(* PLC project CoDeSys External Library Template, WAGO e!COCKPIT e!COCKPIT, author 3S - Smart Software Solutions GmbH *)
(* stored: creationDateTime 2019-10-29T12:22:40.6747974, version 3.5.5.30, modificationDateTime 2019-10-24T14:40:07.960949, organization 3S - Smart Software Solutions GmbH *)
(* Library project template with all possible element types, docu and a sample project structure *)

FUNCTION_BLOCK fbPPPSBramkaSTC65RS485Modbus
  VAR_INPUT
    sKomunikat : alSTRINGKomunikat;  (* komunikat z systemu zewnętrznego *)
    intTablicaKomunikatowRozmiar : INT;  (* rozmiar tablicy danych wysyłkowych *)
    xTablicaKomunikatowHold : BOOL;  (* wstrzymanie komunikacji mniej ważnych komunikatów *)
    sIdInstancji : STRING;  (* parametr ID rolety np NS02L*202IBM**** *)
    sIdAplikacji : STRING;  (* parametr ID aplikacji np SO*******ECL*000 *)
    sMnemonik : STRING;  (* mnemonik właściciela - BCB* *)
    sMACAdres : STRING;  (* MAC adres sterownika *)
    sDaneZapasowe : STRING;  (* 6 znaków zapasu *)
    tCzasOpoznieniaRestartu : TIME;  (* czas opóźnienia po którym zaczynają być raportowane wartości *)
    bAdres : BYTE;
    tMinimalnyCzasRaportowania : TIME;
    tMaksymalnyCzasRaportowania : TIME;
    tCzasTimeoutEnOcean : TIME;
  END_VAR
  VAR_IN_OUT
    arModbusStatusKomunikacji : ARRAY[1..256] OF INT;
    arModbusOdczytCykliczny : ARRAY[1..5000] OF typModbusOdczytCykliczny;
    arTablicaKomunikatow : alARRAYTablicaKomunikatow;
    intTablicaKomunikatowZnacznikZapisu : INT;
  END_VAR
  VAR CONSTANT
    wCzasDzialaniaOdResetuAlarm : WORD := 120;
  END_VAR
  VAR
    xPierwszySkan : BOOL := TRUE;
    intPetlaPierwszySkan : INT := 1;
    xPoInicjalizacji : BOOL := FALSE;  (* inicjalizacja *)
    fbInicjalizacyjnyTimer : TON;
    uintFirmwareVersion : UINT := 0;  (* definicja adresów i zmiennych modbusowych *)
    wFirmwareVersion : WORD;
    uintOperatingTimeSinceLastResetHi : UINT := 2;
    wOperatingTimeSinceLastResetHi : WORD;
    uintOperatingTimeSinceLastResetLo : UINT := 3;
    wOperatingTimeSinceLastResetLo : WORD;
    uintReceivingChannelsTelegramCounterAllIDsHi : UINT := 4;
    wReceivingChannelsTelegramCounterAllIDsHi : WORD;
    uintReceivingChannelsTelegramCounterAllIDsLo : UINT := 5;
    wReceivingChannelsTelegramCounterAllIDsLo : WORD;
    uintReceivingChannelsTelegramCounterStoredIDsHi : UINT := 6;
    wReceivingChannelsTelegramCounterStoredIDsHi : WORD;
    uintReceivingChannelsTelegramCounterStoredIDsLo : UINT := 7;
    wReceivingChannelsTelegramCounterStoredIDsLo : WORD;
    uintEnOceanBaseIdByte3 : UINT := 8;
    wEnOceanBaseIdByte3 : WORD;
    uintEnOceanBaseIdByte2 : UINT := 9;
    wEnOceanBaseIdByte2 : WORD;
    uintEnOceanBaseIdByte1 : UINT := 10;
    wEnOceanBaseIdByte1 : WORD;
    uintEnOceanBaseIdByte0 : UINT := 11;
    wEnOceanBaseIdByte0 : WORD;
    uintRepeaterFunction : UINT := 15;
    wRepeaterFunction : WORD;
    uintMinResponseTime : UINT := 16;
    wMinResponseTime : WORD;
    uintResetRxCoil : UINT := 17;
    wResetRxCoil : WORD;
    uintTransmittingChannelsTelegramCounterAll : UINT := 18;
    wTransmittingChannelsTelegramCounterAll : WORD;
    uintTransmittingChannelsTelegramCounterByCoilTriggered : UINT := 19;
    wTransmittingChannelsTelegramCounterByCoilTriggered : WORD;
    wCzasDzialaniaOdResetuHi : WORD;  (* zmienne operacyjne Zmienne Modbusowe *)
    wCzasDzialaniaOdResetuLo : WORD;
    dwCzasDzialaniaOdResetu : DWORD;
    xAlarmResetu : BOOL;
    wLicznikTelegramowUrzadzenHi : WORD;
    wLicznikTelegramowUrzadzenLo : WORD;
    dwLicznikTelegramowUrzadzen : DWORD;
    dwLicznikTelegramowUrzadzenPamiec : DWORD;
    fbTimeoutEnOcean : TON;
    wFunkcjaPowtarzanaia : WORD;
    wMinimalnyCzasOdpowiedzi : WORD;
    sDane : alSTRINGKomunikat;
    sWyslanyKomunikat : alSTRINGKomunikat;
    sKomunikatPamiec : alSTRINGKomunikat;
    sWyslanyKomunikatDummy : alSTRINGKomunikat;
    intPetla : INT;
    arErrorStan : ARRAY[0..5] OF INT;  (* tablica przechowująca statusy alarmowe *)
    arErrorKlasa : ARRAY[0..5] OF INT;  (* tablica przechowująca klasy danych alarmów *)
    fbBrakKomunikacjiTimer : TON;  (* Wystawianie alarmu o braku komunikacji. Alarm zostanie aktywowany po minutach od momentu stwierdzenia braku komunikacji. *)
  END_VAR

            (*			
Autor:					Paweł Kąkol, 2018-08-13, Jan Bartczak
Prawa majątkowe: 		Solwena Sp. z o.o., 
Aktualizacje:			
						
Opis:					fb służy obsługi bramek (STC65-RS485) GTW0 na budynkach PPP Sopot (ENGIE) 
		
UWAGA:					2018-08-13-PK-Stworzenie FB
						2018-10-05-JB Przygotowanie odczytu rejestrów Modbusowych z bramki STC
						2018-12-11-JB Poprawienie obsługi alarmów od resetu bramki i braku ruchu telegramów (do tego momentu wysyłane były błędne alarmy)		
						2019-02-18-AWy: Filtrowanie alarmu braku komunikacji (5 minut zwłoki od momentu stwierdzenia braku komunikacji)			
*)

//inicjalizacja sterownika
fbInicjalizacyjnyTimer(IN := NOT xPoInicjalizacji , PT := tCzasOpoznieniaRestartu);
IF fbInicjalizacyjnyTimer.Q THEN
	xPoInicjalizacji := TRUE;
	dwLicznikTelegramowUrzadzenPamiec := dwLicznikTelegramowUrzadzen;
END_IF


IF xPierwszySkan THEN
	xPierwszySkan := FALSE;
	WHILE arModbusOdczytCykliczny[intPetlaPierwszySkan].bAdresUrzadzenia <> 0 DO
		intPetlaPierwszySkan := intPetlaPierwszySkan + 1;
	END_WHILE
	
//deklaracja rejestrow do odczytu

	//wyznaczenie adresów rejestrów modbusowych

	//holding register
	//  #Firmware Version e.g.: 0x3300 = Version 3.3.0.0
	arModbusOdczytCykliczny[intPetlaPierwszySkan].bAdresUrzadzenia := bAdres;
	arModbusOdczytCykliczny[intPetlaPierwszySkan].bFunkcja := TO_BYTE(enumModbusKodyFunkcji.OdczytNRejestrow);
	arModbusOdczytCykliczny[intPetlaPierwszySkan].uiAdresRejestru := uintFirmwareVersion;
	arModbusOdczytCykliczny[intPetlaPierwszySkan].ltCzestotliwosc := TIME_TO_LTIME(tMinimalnyCzasRaportowania);
	arModbusOdczytCykliczny[intPetlaPierwszySkan].pZmiennaReferencyjna := ADR(wFirmwareVersion);
	intPetlaPierwszySkan := intPetlaPierwszySkan + 1;

	//R/W Operating Time since last reset [seconds] HIGH
	arModbusOdczytCykliczny[intPetlaPierwszySkan].bAdresUrzadzenia := bAdres;
	arModbusOdczytCykliczny[intPetlaPierwszySkan].bFunkcja := TO_BYTE(enumModbusKodyFunkcji.OdczytNRejestrow);
	arModbusOdczytCykliczny[intPetlaPierwszySkan].uiAdresRejestru := uintOperatingTimeSinceLastResetHi;
	arModbusOdczytCykliczny[intPetlaPierwszySkan].ltCzestotliwosc := TIME_TO_LTIME(tMinimalnyCzasRaportowania);
	arModbusOdczytCykliczny[intPetlaPierwszySkan].pZmiennaReferencyjna := ADR(wOperatingTimeSinceLastResetHi);
	intPetlaPierwszySkan := intPetlaPierwszySkan + 1;	
	
	//R/W Operating Time since last reset [seconds] LOW
	arModbusOdczytCykliczny[intPetlaPierwszySkan].bAdresUrzadzenia := bAdres;
	arModbusOdczytCykliczny[intPetlaPierwszySkan].bFunkcja := TO_BYTE(enumModbusKodyFunkcji.OdczytNRejestrow);
	arModbusOdczytCykliczny[intPetlaPierwszySkan].uiAdresRejestru := uintOperatingTimeSinceLastResetLo;
	arModbusOdczytCykliczny[intPetlaPierwszySkan].ltCzestotliwosc := TIME_TO_LTIME(tMinimalnyCzasRaportowania);
	arModbusOdczytCykliczny[intPetlaPierwszySkan].pZmiennaReferencyjna := ADR(wOperatingTimeSinceLastResetLo);
	intPetlaPierwszySkan := intPetlaPierwszySkan + 1;	
	
	//R/W Receiving Channels Telegram Counter (all IDs) HIGH
	arModbusOdczytCykliczny[intPetlaPierwszySkan].bAdresUrzadzenia := bAdres;
	arModbusOdczytCykliczny[intPetlaPierwszySkan].bFunkcja := TO_BYTE(enumModbusKodyFunkcji.OdczytNRejestrow);
	arModbusOdczytCykliczny[intPetlaPierwszySkan].uiAdresRejestru := uintReceivingChannelsTelegramCounterAllIDsHi;
	arModbusOdczytCykliczny[intPetlaPierwszySkan].ltCzestotliwosc := TIME_TO_LTIME(tMinimalnyCzasRaportowania);
	arModbusOdczytCykliczny[intPetlaPierwszySkan].pZmiennaReferencyjna := ADR(wReceivingChannelsTelegramCounterAllIDsHi);
	intPetlaPierwszySkan := intPetlaPierwszySkan + 1;		

	//R/W Receiving Channels Telegram Counter (all IDs) LOW	
	arModbusOdczytCykliczny[intPetlaPierwszySkan].bAdresUrzadzenia := bAdres;
	arModbusOdczytCykliczny[intPetlaPierwszySkan].bFunkcja := TO_BYTE(enumModbusKodyFunkcji.OdczytNRejestrow);
	arModbusOdczytCykliczny[intPetlaPierwszySkan].uiAdresRejestru := uintReceivingChannelsTelegramCounterAllIDsLo;
	arModbusOdczytCykliczny[intPetlaPierwszySkan].ltCzestotliwosc := TIME_TO_LTIME(tMinimalnyCzasRaportowania);
	arModbusOdczytCykliczny[intPetlaPierwszySkan].pZmiennaReferencyjna := ADR(wReceivingChannelsTelegramCounterAllIDsLo);
	intPetlaPierwszySkan := intPetlaPierwszySkan + 1;

	//R/W Receiving Channels Telegram Counter (stored IDs only) HIGH
	arModbusOdczytCykliczny[intPetlaPierwszySkan].bAdresUrzadzenia := bAdres;
	arModbusOdczytCykliczny[intPetlaPierwszySkan].bFunkcja := TO_BYTE(enumModbusKodyFunkcji.OdczytNRejestrow);
	arModbusOdczytCykliczny[intPetlaPierwszySkan].uiAdresRejestru := uintReceivingChannelsTelegramCounterStoredIDsHi;
	arModbusOdczytCykliczny[intPetlaPierwszySkan].ltCzestotliwosc := TIME_TO_LTIME(tMinimalnyCzasRaportowania);
	arModbusOdczytCykliczny[intPetlaPierwszySkan].pZmiennaReferencyjna := ADR(wReceivingChannelsTelegramCounterStoredIDsHi);
	intPetlaPierwszySkan := intPetlaPierwszySkan + 1;

	//R/W Receiving Channels Telegram Counter (stored IDs only) LOW
	arModbusOdczytCykliczny[intPetlaPierwszySkan].bAdresUrzadzenia := bAdres;
	arModbusOdczytCykliczny[intPetlaPierwszySkan].bFunkcja := TO_BYTE(enumModbusKodyFunkcji.OdczytNRejestrow);
	arModbusOdczytCykliczny[intPetlaPierwszySkan].uiAdresRejestru := uintReceivingChannelsTelegramCounterStoredIDsLo;
	arModbusOdczytCykliczny[intPetlaPierwszySkan].ltCzestotliwosc := TIME_TO_LTIME(tMinimalnyCzasRaportowania);
	arModbusOdczytCykliczny[intPetlaPierwszySkan].pZmiennaReferencyjna := ADR(wReceivingChannelsTelegramCounterStoredIDsLo);
	intPetlaPierwszySkan := intPetlaPierwszySkan + 1;	
	
	//R/W* #EnOcean Base-ID-Byte-3
	arModbusOdczytCykliczny[intPetlaPierwszySkan].bAdresUrzadzenia := bAdres;
	arModbusOdczytCykliczny[intPetlaPierwszySkan].bFunkcja := TO_BYTE(enumModbusKodyFunkcji.OdczytNRejestrow);
	arModbusOdczytCykliczny[intPetlaPierwszySkan].uiAdresRejestru := uintEnOceanBaseIdByte3;
	arModbusOdczytCykliczny[intPetlaPierwszySkan].ltCzestotliwosc := TIME_TO_LTIME(tMinimalnyCzasRaportowania);
	arModbusOdczytCykliczny[intPetlaPierwszySkan].pZmiennaReferencyjna := ADR(wEnOceanBaseIdByte3);
	intPetlaPierwszySkan := intPetlaPierwszySkan + 1;	
	
	//R/W* #EnOcean Base-ID-Byte-2
	arModbusOdczytCykliczny[intPetlaPierwszySkan].bAdresUrzadzenia := bAdres;
	arModbusOdczytCykliczny[intPetlaPierwszySkan].bFunkcja := TO_BYTE(enumModbusKodyFunkcji.OdczytNRejestrow);
	arModbusOdczytCykliczny[intPetlaPierwszySkan].uiAdresRejestru := uintEnOceanBaseIdByte2;
	arModbusOdczytCykliczny[intPetlaPierwszySkan].ltCzestotliwosc := TIME_TO_LTIME(tMinimalnyCzasRaportowania);
	arModbusOdczytCykliczny[intPetlaPierwszySkan].pZmiennaReferencyjna := ADR(wEnOceanBaseIdByte2);
	intPetlaPierwszySkan := intPetlaPierwszySkan + 1;		

	//R/W* #EnOcean Base-ID-Byte-1
	arModbusOdczytCykliczny[intPetlaPierwszySkan].bAdresUrzadzenia := bAdres;
	arModbusOdczytCykliczny[intPetlaPierwszySkan].bFunkcja := TO_BYTE(enumModbusKodyFunkcji.OdczytNRejestrow);
	arModbusOdczytCykliczny[intPetlaPierwszySkan].uiAdresRejestru := uintEnOceanBaseIdByte1;
	arModbusOdczytCykliczny[intPetlaPierwszySkan].ltCzestotliwosc := TIME_TO_LTIME(tMinimalnyCzasRaportowania);
	arModbusOdczytCykliczny[intPetlaPierwszySkan].pZmiennaReferencyjna := ADR(wEnOceanBaseIdByte1);
	intPetlaPierwszySkan := intPetlaPierwszySkan + 1;		

	//R/W* #EnOcean Base-ID-Byte-0
	arModbusOdczytCykliczny[intPetlaPierwszySkan].bAdresUrzadzenia := bAdres;
	arModbusOdczytCykliczny[intPetlaPierwszySkan].bFunkcja := TO_BYTE(enumModbusKodyFunkcji.OdczytNRejestrow);
	arModbusOdczytCykliczny[intPetlaPierwszySkan].uiAdresRejestru := uintEnOceanBaseIdByte0;
	arModbusOdczytCykliczny[intPetlaPierwszySkan].ltCzestotliwosc := TIME_TO_LTIME(tMinimalnyCzasRaportowania);
	arModbusOdczytCykliczny[intPetlaPierwszySkan].pZmiennaReferencyjna := ADR(wEnOceanBaseIdByte0);
	intPetlaPierwszySkan := intPetlaPierwszySkan + 1;		
	
	//#Repeater function (0=OFF, 1=1-Level, 2=2-Level) ; Sets the integrated EnOcean repeater to off, 1-level or 2-level
	arModbusOdczytCykliczny[intPetlaPierwszySkan].bAdresUrzadzenia := bAdres;
	arModbusOdczytCykliczny[intPetlaPierwszySkan].bFunkcja := TO_BYTE(enumModbusKodyFunkcji.OdczytNRejestrow);
	arModbusOdczytCykliczny[intPetlaPierwszySkan].uiAdresRejestru := uintRepeaterFunction;
	arModbusOdczytCykliczny[intPetlaPierwszySkan].ltCzestotliwosc := TIME_TO_LTIME(tMinimalnyCzasRaportowania);
	arModbusOdczytCykliczny[intPetlaPierwszySkan].pZmiennaReferencyjna := ADR(wRepeaterFunction);
	intPetlaPierwszySkan := intPetlaPierwszySkan + 1;			
	
	//R/W #Min. Response Time 
	arModbusOdczytCykliczny[intPetlaPierwszySkan].bAdresUrzadzenia := bAdres;
	arModbusOdczytCykliczny[intPetlaPierwszySkan].bFunkcja := TO_BYTE(enumModbusKodyFunkcji.OdczytNRejestrow);
	arModbusOdczytCykliczny[intPetlaPierwszySkan].uiAdresRejestru := uintMinResponseTime;
	arModbusOdczytCykliczny[intPetlaPierwszySkan].ltCzestotliwosc := TIME_TO_LTIME(tMinimalnyCzasRaportowania);
	arModbusOdczytCykliczny[intPetlaPierwszySkan].pZmiennaReferencyjna := ADR(wMinResponseTime);
	intPetlaPierwszySkan := intPetlaPierwszySkan + 1;		
	
	//R/W #Reset RX Coil necessary (factory setting: 0)
	arModbusOdczytCykliczny[intPetlaPierwszySkan].bAdresUrzadzenia := bAdres;
	arModbusOdczytCykliczny[intPetlaPierwszySkan].bFunkcja := TO_BYTE(enumModbusKodyFunkcji.OdczytNRejestrow);
	arModbusOdczytCykliczny[intPetlaPierwszySkan].uiAdresRejestru := uintResetRxCoil;
	arModbusOdczytCykliczny[intPetlaPierwszySkan].ltCzestotliwosc := TIME_TO_LTIME(tMinimalnyCzasRaportowania);
	arModbusOdczytCykliczny[intPetlaPierwszySkan].pZmiennaReferencyjna := ADR(wResetRxCoil);
	intPetlaPierwszySkan := intPetlaPierwszySkan + 1;		
	
	//R/W Transmitting Channels Telegram Counter (all telegrams)
	arModbusOdczytCykliczny[intPetlaPierwszySkan].bAdresUrzadzenia := bAdres;
	arModbusOdczytCykliczny[intPetlaPierwszySkan].bFunkcja := TO_BYTE(enumModbusKodyFunkcji.OdczytNRejestrow);
	arModbusOdczytCykliczny[intPetlaPierwszySkan].uiAdresRejestru := uintTransmittingChannelsTelegramCounterAll;
	arModbusOdczytCykliczny[intPetlaPierwszySkan].ltCzestotliwosc := TIME_TO_LTIME(tMinimalnyCzasRaportowania);
	arModbusOdczytCykliczny[intPetlaPierwszySkan].pZmiennaReferencyjna := ADR(wTransmittingChannelsTelegramCounterAll);
	intPetlaPierwszySkan := intPetlaPierwszySkan + 1;	

	//R/W Transmitting Channels Telegram Counter (by coil triggered telegrams only)
	arModbusOdczytCykliczny[intPetlaPierwszySkan].bAdresUrzadzenia := bAdres;
	arModbusOdczytCykliczny[intPetlaPierwszySkan].bFunkcja := TO_BYTE(enumModbusKodyFunkcji.OdczytNRejestrow);
	arModbusOdczytCykliczny[intPetlaPierwszySkan].uiAdresRejestru := uintTransmittingChannelsTelegramCounterByCoilTriggered;
	arModbusOdczytCykliczny[intPetlaPierwszySkan].ltCzestotliwosc := TIME_TO_LTIME(tMinimalnyCzasRaportowania);
	arModbusOdczytCykliczny[intPetlaPierwszySkan].pZmiennaReferencyjna := ADR(wTransmittingChannelsTelegramCounterByCoilTriggered);
	intPetlaPierwszySkan := intPetlaPierwszySkan + 1;	
END_IF

//obsluga komunikatu przychodzacego z IZE

IF 	sKomunikat <> sKomunikatPamiec AND xPoInicjalizacji THEN
	sKomunikatPamiec := sKomunikat;
	IF fnIDOdbiorcyMatch(sKomunikat , sIdInstancji) THEN
		sDane := '';
		//zapytanie typu Q
		IF fnKomunikatTyp(sKomunikat) = 'Q' THEN
			//pytanie o stany alarmów
			IF fnKomunikatDaneSzukajWartosci(sKomunikat , 'ALARM=') = '?' OR fnKomunikatDaneSzukajWartosci(sKomunikat , 'ALL=') = '?' THEN
				FOR intPetla := 1 TO 5 BY 1 DO
					//raportowanie typu E (stanów alarmów) na zapytanie typu Q
					IF arErrorStan[intPetla] <> enumAlarmWartosc.StanNieznany THEN
						fnZapiszKomunikat(	sCalyKomunikat := '' ,
											sTypKomunikatu := 'E' ,
											sMnemonik := sMnemonik ,
											sMACAdres := sMACAdres ,
											sIDNadawcy := sIdInstancji ,
											sIDOdbiorcy := sIdAplikacji ,
											sDaneZapasowe := sDaneZapasowe ,
											sDane := fnKomunikatDaneErrorRetry(xAktywny := arErrorStan[intPetla] = enumAlarmWartosc.StanAlarmowy , intKlasa := arErrorKlasa[intPetla] , intNumer := intPetla),
											arTablicaKomunikatow := arTablicaKomunikatow ,
											intTablicaKomunikatowZnacznikZapisu := intTablicaKomunikatowZnacznikZapisu ,
											intTablicaKomunikatowRozmiar := intTablicaKomunikatowRozmiar ,
											sWyslanyKomunikat := sWyslanyKomunikatDummy);
					END_IF
				END_FOR
			END_IF
		END_IF
		//raportowanie typu A na zapytanie Q
		IF sDane <> '' THEN
			fnZapiszKomunikat(	sCalyKomunikat := '' ,
								sTypKomunikatu := 'A' ,
								sMnemonik := sMnemonik ,
								sMACAdres := sMACAdres ,
								sIDNadawcy := sIdInstancji ,
								sIDOdbiorcy := sIdAplikacji ,
								sDaneZapasowe := sDaneZapasowe ,
								sDane := sDane ,
								arTablicaKomunikatow := arTablicaKomunikatow ,
								intTablicaKomunikatowZnacznikZapisu := intTablicaKomunikatowZnacznikZapisu ,
								intTablicaKomunikatowRozmiar := intTablicaKomunikatowRozmiar ,
								sWyslanyKomunikat := sWyslanyKomunikatDummy);
		END_IF
	END_IF
END_IF

//obliczenia
dwCzasDzialaniaOdResetu := wOperatingTimeSinceLastResetHi * 256 * 256 + wOperatingTimeSinceLastResetLo;
IF dwCzasDzialaniaOdResetu > 0 THEN
	IF dwCzasDzialaniaOdResetu < WORD_TO_DWORD(wCzasDzialaniaOdResetuAlarm) THEN
		xAlarmResetu := TRUE;
	ELSE
		IF dwCzasDzialaniaOdResetu > WORD_TO_DWORD(wCzasDzialaniaOdResetuAlarm) THEN
			xAlarmResetu := FALSE;
		END_IF
	END_IF
END_IF

dwLicznikTelegramowUrzadzen := wReceivingChannelsTelegramCounterAllIDsHi * 256 * 256 + wReceivingChannelsTelegramCounterAllIDsLo;
IF xPoInicjalizacji THEN
	fbTimeoutEnOcean(IN := (dwLicznikTelegramowUrzadzen = dwLicznikTelegramowUrzadzenPamiec) , PT := tCzasTimeoutEnOcean);
END_IF

IF dwLicznikTelegramowUrzadzen <> dwLicznikTelegramowUrzadzenPamiec THEN
	dwLicznikTelegramowUrzadzenPamiec := dwLicznikTelegramowUrzadzen;
END_IF

// Filtrowanie alarmu o braku komunikacji. Alarm wystąpi po 5 minutach od momentu wystąpienia arModbusStatusKomunikacji[bAdres] = enumModbusStatus.BrakKomunikacji
fbBrakKomunikacjiTimer(IN := arModbusStatusKomunikacji[bAdres] = enumModbusStatus.BrakKomunikacji, PT := T#5M);

// obsługa alarmów konwertera
	//brak komunikacji
IF arErrorStan[enumPPPSBramkaSTC65RS485ModbusError.BrakKomunikacji] <> enumAlarmWartosc.StanAlarmowy AND fbBrakKomunikacjiTimer.Q THEN
	arErrorStan[enumPPPSBramkaSTC65RS485ModbusError.BrakKomunikacji] := enumAlarmWartosc.StanAlarmowy;
	arErrorKlasa[enumPPPSBramkaSTC65RS485ModbusError.BrakKomunikacji] :=enumPPPSBramkaSTC65RS485ModbusErrorKlasa.BrakKomunikacji;
	IF xPoInicjalizacji THEN
		fnZapiszKomunikat(	sCalyKomunikat := '' ,
							sTypKomunikatu := 'E' ,
							sMnemonik := sMnemonik ,
							sMACAdres := sMACAdres ,
							sIDNadawcy := sIdInstancji ,
							sIDOdbiorcy := sIdAplikacji ,
							sDaneZapasowe := sDaneZapasowe ,
							sDane := fnKomunikatDaneError(xAktywny := TRUE , intKlasa := enumPPPSBramkaSTC65RS485ModbusErrorKlasa.BrakKomunikacji , intNumer := enumPPPSBramkaSTC65RS485ModbusError.BrakKomunikacji),
							arTablicaKomunikatow := arTablicaKomunikatow ,
							intTablicaKomunikatowZnacznikZapisu := intTablicaKomunikatowZnacznikZapisu ,
							intTablicaKomunikatowRozmiar := intTablicaKomunikatowRozmiar ,
							sWyslanyKomunikat := sWyslanyKomunikatDummy);
	END_IF
END_IF
IF arErrorStan[enumPPPSBramkaSTC65RS485ModbusError.BrakKomunikacji] <> enumAlarmWartosc.StanNormalny AND NOT fbBrakKomunikacjiTimer.Q  THEN
	arErrorStan[enumPPPSBramkaSTC65RS485ModbusError.BrakKomunikacji] := enumAlarmWartosc.StanNormalny;
	arErrorKlasa[enumPPPSBramkaSTC65RS485ModbusError.BrakKomunikacji] := enumPPPSBramkaSTC65RS485ModbusErrorKlasa.BrakKomunikacji;
	IF xPoInicjalizacji THEN
		fnZapiszKomunikat(	sCalyKomunikat := '' ,
							sTypKomunikatu := 'E' ,
							sMnemonik := sMnemonik ,
							sMACAdres := sMACAdres ,
							sIDNadawcy := sIdInstancji ,
							sIDOdbiorcy := sIdAplikacji ,
							sDaneZapasowe := sDaneZapasowe ,
							sDane := fnKomunikatDaneError(xAktywny := FALSE , intKlasa := enumPPPSBramkaSTC65RS485ModbusErrorKlasa.BrakKomunikacji , intNumer := enumPPPSBramkaSTC65RS485ModbusError.BrakKomunikacji),
							arTablicaKomunikatow := arTablicaKomunikatow ,
							intTablicaKomunikatowZnacznikZapisu := intTablicaKomunikatowZnacznikZapisu ,
							intTablicaKomunikatowRozmiar := intTablicaKomunikatowRozmiar ,
							sWyslanyKomunikat := sWyslanyKomunikatDummy);
	END_IF
END_IF

	//reset konwertera
IF arErrorStan[enumPPPSBramkaSTC65RS485ModbusError.ResetKonwertera] <> enumAlarmWartosc.StanAlarmowy AND xAlarmResetu AND arModbusStatusKomunikacji[bAdres] = enumModbusStatus.KomunikacjaPrawidlowa THEN
	arErrorStan[enumPPPSBramkaSTC65RS485ModbusError.ResetKonwertera] := enumAlarmWartosc.StanAlarmowy;
	arErrorKlasa[enumPPPSBramkaSTC65RS485ModbusError.ResetKonwertera] :=enumPPPSBramkaSTC65RS485ModbusErrorKlasa.ResetKonwertera;
	IF xPoInicjalizacji THEN
		fnZapiszKomunikat(	sCalyKomunikat := '' ,
							sTypKomunikatu := 'E' ,
							sMnemonik := sMnemonik ,
							sMACAdres := sMACAdres ,
							sIDNadawcy := sIdInstancji ,
							sIDOdbiorcy := sIdAplikacji ,
							sDaneZapasowe := sDaneZapasowe ,
							sDane := fnKomunikatDaneError(xAktywny := TRUE , intKlasa := enumPPPSBramkaSTC65RS485ModbusErrorKlasa.ResetKonwertera , intNumer := enumPPPSBramkaSTC65RS485ModbusError.ResetKonwertera),
							arTablicaKomunikatow := arTablicaKomunikatow ,
							intTablicaKomunikatowZnacznikZapisu := intTablicaKomunikatowZnacznikZapisu ,
							intTablicaKomunikatowRozmiar := intTablicaKomunikatowRozmiar ,
							sWyslanyKomunikat := sWyslanyKomunikatDummy);
	END_IF
END_IF
IF arErrorStan[enumPPPSBramkaSTC65RS485ModbusError.ResetKonwertera] <> enumAlarmWartosc.StanNormalny AND NOT xAlarmResetu AND arModbusStatusKomunikacji[bAdres] = enumModbusStatus.KomunikacjaPrawidlowa THEN
	arErrorStan[enumPPPSBramkaSTC65RS485ModbusError.ResetKonwertera] := enumAlarmWartosc.StanNormalny;
	arErrorKlasa[enumPPPSBramkaSTC65RS485ModbusError.ResetKonwertera] := enumPPPSBramkaSTC65RS485ModbusErrorKlasa.ResetKonwertera;
	IF xPoInicjalizacji THEN
		fnZapiszKomunikat(	sCalyKomunikat := '' ,
							sTypKomunikatu := 'E' ,
							sMnemonik := sMnemonik ,
							sMACAdres := sMACAdres ,
							sIDNadawcy := sIdInstancji ,
							sIDOdbiorcy := sIdAplikacji ,
							sDaneZapasowe := sDaneZapasowe ,
							sDane := fnKomunikatDaneError(xAktywny := FALSE , intKlasa := enumPPPSBramkaSTC65RS485ModbusErrorKlasa.ResetKonwertera , intNumer := enumPPPSBramkaSTC65RS485ModbusError.ResetKonwertera),
							arTablicaKomunikatow := arTablicaKomunikatow ,
							intTablicaKomunikatowZnacznikZapisu := intTablicaKomunikatowZnacznikZapisu ,
							intTablicaKomunikatowRozmiar := intTablicaKomunikatowRozmiar ,
							sWyslanyKomunikat := sWyslanyKomunikatDummy);
	END_IF
END_IF

	//brak telegramów
IF arErrorStan[enumPPPSBramkaSTC65RS485ModbusError.BrakTelegramowEnOcean] <> enumAlarmWartosc.StanAlarmowy AND fbTimeoutEnOcean.Q AND arModbusStatusKomunikacji[bAdres] = enumModbusStatus.KomunikacjaPrawidlowa THEN
	arErrorStan[enumPPPSBramkaSTC65RS485ModbusError.BrakTelegramowEnOcean] := enumAlarmWartosc.StanAlarmowy;
	arErrorKlasa[enumPPPSBramkaSTC65RS485ModbusError.BrakTelegramowEnOcean] :=enumPPPSBramkaSTC65RS485ModbusErrorKlasa.BrakTelegramowEnOcean;
	IF xPoInicjalizacji THEN
		fnZapiszKomunikat(	sCalyKomunikat := '' ,
							sTypKomunikatu := 'E' ,
							sMnemonik := sMnemonik ,
							sMACAdres := sMACAdres ,
							sIDNadawcy := sIdInstancji ,
							sIDOdbiorcy := sIdAplikacji ,
							sDaneZapasowe := sDaneZapasowe ,
							sDane := fnKomunikatDaneError(xAktywny := TRUE , intKlasa := enumPPPSBramkaSTC65RS485ModbusErrorKlasa.BrakTelegramowEnOcean , intNumer := enumPPPSBramkaSTC65RS485ModbusError.BrakTelegramowEnOcean),
							arTablicaKomunikatow := arTablicaKomunikatow ,
							intTablicaKomunikatowZnacznikZapisu := intTablicaKomunikatowZnacznikZapisu ,
							intTablicaKomunikatowRozmiar := intTablicaKomunikatowRozmiar ,
							sWyslanyKomunikat := sWyslanyKomunikatDummy);
	END_IF
END_IF
IF arErrorStan[enumPPPSBramkaSTC65RS485ModbusError.BrakTelegramowEnOcean] <> enumAlarmWartosc.StanNormalny AND NOT fbTimeoutEnOcean.Q AND arModbusStatusKomunikacji[bAdres] = enumModbusStatus.KomunikacjaPrawidlowa THEN
	arErrorStan[enumPPPSBramkaSTC65RS485ModbusError.BrakTelegramowEnOcean] := enumAlarmWartosc.StanNormalny;
	arErrorKlasa[enumPPPSBramkaSTC65RS485ModbusError.BrakTelegramowEnOcean] := enumPPPSBramkaSTC65RS485ModbusErrorKlasa.BrakTelegramowEnOcean;
	IF xPoInicjalizacji THEN
		fnZapiszKomunikat(	sCalyKomunikat := '' ,
							sTypKomunikatu := 'E' ,
							sMnemonik := sMnemonik ,
							sMACAdres := sMACAdres ,
							sIDNadawcy := sIdInstancji ,
							sIDOdbiorcy := sIdAplikacji ,
							sDaneZapasowe := sDaneZapasowe ,
							sDane := fnKomunikatDaneError(xAktywny := FALSE , intKlasa := enumPPPSBramkaSTC65RS485ModbusErrorKlasa.BrakTelegramowEnOcean , intNumer := enumPPPSBramkaSTC65RS485ModbusError.BrakTelegramowEnOcean),
							arTablicaKomunikatow := arTablicaKomunikatow ,
							intTablicaKomunikatowZnacznikZapisu := intTablicaKomunikatowZnacznikZapisu ,
							intTablicaKomunikatowRozmiar := intTablicaKomunikatowRozmiar ,
							sWyslanyKomunikat := sWyslanyKomunikatDummy);
	END_IF
END_IF


          
END_FUNCTION_BLOCK
